FUNCTION F_PHYS_TO_RAW (* Convert physical REAL value to ISOBUS raw UDINT with saturation and alarm outputs. ISOBUS formula: display = (raw + offset) * scale Inverse: raw = UDINT(DINT(phys / scale) - offset) Limits: phys < offset * scale          -> udRaw = 0,           xUnder = TRUE phys > (offset + 4294967295) * scale -> udRaw = UDINT#MAX,   xOver = TRUE Example: phys=-500.0, scale=0.01, offset=-100000 DINT(-500.0 / 0.01) = -50000 -50000 - (-100000) = 50000 UDINT(50000) = 50000 -> UT displays (50000 + (-100000)) * 0.01 = -500.00 *)
  (* Standard: 61499-2; Description: Copyright (c) 2026 Meisterschulen am Ostbahnhof This program and the accompanying materials are made available under the terms of the Eclipse Public License 2.0 which is available at https://www.eclipse.org/legal/epl-2.0/ SPDX-License-Identifier: EPL-2.0 *)
  (* Version 1.0, 2026-04-14, Franz Höpfinger, Meisterschulen am Ostbahnhof *)
  PACKAGE logiBUS::utils::conversion::phys;
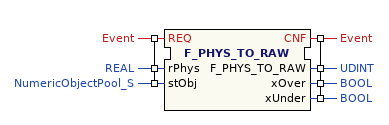
  EVENT_INPUT
    REQ WITH rPhys, stObj;
  END_EVENT
  EVENT_OUTPUT
    CNF WITH F_PHYS_TO_RAW, xOver, xUnder;
  END_EVENT
  VAR_INPUT
    rPhys : REAL;
    stObj : logiBUS::utils::conversion::phys::NumericObjectPool_S;
  END_VAR
  VAR_OUTPUT
    F_PHYS_TO_RAW : UDINT;
    xOver : BOOL;
    xUnder : BOOL;
  END_VAR
  BODY IN ST:
PACKAGE logiBUS::utils::conversion::phys;

(* Convert physical REAL value to ISOBUS raw UDINT with saturation and alarm outputs.
 * ISOBUS formula: display = (raw + offset) * scale
 * Inverse: raw = UDINT(DINT(phys / scale) - offset)
 *
 * Limits:
 *   phys < offset * scale          -> udRaw = 0,           xUnder = TRUE
 *   phys > (offset + 4294967295) * scale -> udRaw = UDINT#MAX,   xOver = TRUE
 *
 * Example: phys=-500.0, scale=0.01, offset=-100000
 *   DINT(-500.0 / 0.01) = -50000
 *   -50000 - (-100000) = 50000
 *   UDINT(50000) = 50000 -> UT displays (50000 + (-100000)) * 0.01 = -500.00 *)
FUNCTION F_PHYS_TO_RAW : UDINT

VAR_INPUT
	rPhys : REAL;
	stObj : NumericObjectPool_S;
END_VAR

VAR_OUTPUT
	xOver : BOOL;
	xUnder : BOOL;
END_VAR

VAR
	lrLower : REAL;
	lrUpper : REAL;
END_VAR

lrLower := DINT_TO_REAL(stObj.i32Offset) * stObj.r32Scale;
lrUpper := (DINT_TO_REAL(stObj.i32Offset) + REAL#4294967295.0) * stObj.r32Scale;

IF rPhys > lrUpper THEN
	F_PHYS_TO_RAW := UDINT#4294967295;
	xOver := TRUE;
	xUnder := FALSE;
ELSIF rPhys < lrLower THEN
	F_PHYS_TO_RAW := UDINT#0;
	xOver := FALSE;
	xUnder := TRUE;
ELSE
	F_PHYS_TO_RAW := DINT_TO_UDINT(REAL_TO_DINT(rPhys / stObj.r32Scale) - stObj.i32Offset);
	xOver := FALSE;
	xUnder := FALSE;
END_IF;

END_FUNCTION
  END_BODY
END_FUNCTION
